// TwinCAT 3 PLC project SAT_Bibliothek
// Title: STOBER_G6_Util
// Company: STÖBER Antriebstechnik GmbH + Co. KG
// Author: STOBER
// ProjectVersion: 3.1.1.0
// Description: The function blocks in the library would be operational with STOBER drive controller Firmware version 6.5-F and higher.
// ProgramVersion: 3.1.4024.12
// libraries:
//   Tc2_EtherCAT, * (Beckhoff Automation GmbH)
//   Tc2_MC2, * (Beckhoff Automation GmbH)
//   Tc2_MC2_Drive, * (Beckhoff Automation GmbH)
//   Tc2_Standard, * (Beckhoff Automation GmbH)
//   Tc2_System, * (Beckhoff Automation GmbH)
//   Tc2_Utilities, * (Beckhoff Automation GmbH)
//   Tc3_Module, * (Beckhoff Automation GmbH)
// project tree:
//   DUTs/STOBER_Backup_Restore/ eFBERROR.TcTLEO, eSERVICE.TcTLEO, eWriteState.TcTLEO, E_EventType.TcTLEO, ST_DeviceInfo.TcDUT, ST_Event.TcDUT
//   DUTs/STOBER_Boxname/ Ethercat_State.TcDUT, StoeberSlavedesc.TcDUT, St_Error.TcDUT
//   DUTs/STOBER_MC_HOME/ eERROR.TcTLEO, st_Set_Value.TcDUT
//   GVLs/ GLOBAL_DeviceInfo.TcGVL, GVL_Constant.TcGVL
//   POUs/ FB_STOBER_BASE.TcPOU, STOBER_Backup_Restore.TcPOU, STOBER_BoxName.TcPOU, STOBER_MC_HOME.TcPOU
//   POUs/Functions/ CONCAT4.TcPOU, CONCAT8.TcPOU
//   POUs/Logger/ FB_logger.TcPOU, FB_LogPersistentStorage.TcPOU, GetSystemTimeStamp.TcPOU, I_PersistentEventStorage.TcIO
//   Project Information/ F_GetCompany.TcPOU, F_GetTitle.TcPOU, F_GetVersion.TcPOU
//   Version/ Global_Version.TcGVL

// ---- DUTs/STOBER_Backup_Restore/eFBERROR.TcTLEO
{attribute 'qualified_only'}
{attribute 'strict'}
TYPE eFBERROR :
(   
	(*Function block errors*)
	NoError								:=0,
	WrongFilePath						:=101,
	WrongDS6_ProcessPath				:=103,
	WrongEtherCATRevision				:=105,
	InvalidBoxname						:=107,
	WrongServiceTypeInput				:=109,
	TimeoutExceed						:=111,
	NoStoberSlaveInConfiguration		:=113,
	
	(*DS6 Errors*)
	ProjectNotFound						:=201,//Drive controller project not found
	MoreThanOneProjectFound				:=203,//Drive Controller found several times in project 
	OpenProjectError					:=205,//project open error 
	ConnectionError						:=207,//Connection to Drive controller failed 
	OnlineError							:=209//Online connection failed 
	
	


);
END_TYPE

// ---- DUTs/STOBER_Backup_Restore/eSERVICE.TcTLEO
{attribute 'qualified_only'}
{attribute 'strict'}
TYPE eSERVICE :
(
	Backup			:=0,
	Backup_RevDocu	:=1,
	Restore			:=2

);
END_TYPE

// ---- DUTs/STOBER_Backup_Restore/eWriteState.TcTLEO
{attribute 'qualified_only'}
{attribute 'strict'}
{attribute  'hide'}
TYPE eWriteState :
(
	FileOpen_TRIGGER,
	FILE_OPEN,
	WAIT_FOR_EVENT,
	WRITE_EVENT_TRIGGER,
	WRITE_EVENT,
	FILE_CLOSE_TRIGGER,
	FILE_CLOSE,ERROR
);
END_TYPE

// ---- DUTs/STOBER_Backup_Restore/E_EventType.TcTLEO
{attribute 'qualified_only'}
{attribute 'strict'}
{attribute 'to_string'}
{attribute  'hide'}
TYPE E_EventType :
(
	Info:=0,
	Warning:=1,
	Error:=2
);
END_TYPE

// ---- DUTs/STOBER_Backup_Restore/ST_DeviceInfo.TcDUT
{attribute  'hide'}
TYPE ST_DeviceInfo :
STRUCT
	Slave_Address		:STRING(16);
	Production_Number	:STRING(16);
END_STRUCT
END_TYPE

// ---- DUTs/STOBER_Backup_Restore/ST_Event.TcDUT
{attribute  'hide'}
TYPE ST_Event :
STRUCT
	EventType:T_MaxString;
	sEventText:T_MaxString;
	timesatamp:T_MaxString;
END_STRUCT
END_TYPE

// ---- DUTs/STOBER_Boxname/Ethercat_State.TcDUT
{attribute 'qualified_only'}
{attribute 'strict'}
{attribute 'hide'}
TYPE Ethercat_State :
(
	INIT :=1,
	PREOP:=2,
	SAFEOP:=4,
	OP:=8
);
END_TYPE

// ---- DUTs/STOBER_Boxname/StoeberSlavedesc.TcDUT
{attribute 'hide'}
TYPE StoeberSlavedesc :
STRUCT
	nAddr:WORD;
	sType:STRING(15);
	{attribute 'TcEncoding' := 'UTF-8'}
	sName:STRING(31);
	nDevType:DWORD;
	iState:INT;
END_STRUCT
END_TYPE

// ---- DUTs/STOBER_Boxname/St_Error.TcDUT
{attribute 'hide'}
TYPE St_Error :
STRUCT
	
END_STRUCT
END_TYPE

// ---- DUTs/STOBER_MC_HOME/eERROR.TcTLEO
{attribute 'qualified_only'}
{attribute 'strict'}
TYPE eERROR :
(
	NO_ERROR := 0, //Defined operation was executed successfully
	HOMING_METHOD_INACTIVE:=1,//NO homing method selected 
	AXIS_NOT_ENABLED:=2,//Axis is not enabled 
	WRONG_MODE:=3,//Wrong mode of operation input 
	NO_DEVICE_LINK:=4//ModeOfOperation output variable is not linked in device config  
);
END_TYPE

// ---- DUTs/STOBER_MC_HOME/st_Set_Value.TcDUT
{attribute 'hide'}
TYPE st_Set_Value :
STRUCT
	SetPosition		:LREAL;
	SetVelocity		:LREAL;
	SetAcc			:LREAL;
	SetDec			:LREAL;
	SetDirection	:LREAL;
	SetJerk			:LREAL;
END_STRUCT
END_TYPE

// ---- GVLs/GLOBAL_DeviceInfo.TcGVL
{attribute 'qualified_only'}
VAR_GLOBAL
	arr_DeviceInfodata:ARRAY [1..GVL_Constant.MAX_STOBER_SLAVES] OF ST_DeviceInfo;
END_VAR

// ---- GVLs/GVL_Constant.TcGVL
{attribute 'qualified_only'}
VAR_GLOBAL CONSTANT
	MAX_STOBER_SLAVES:INT:=200;
	MaxSlaves:INT:=2000;
END_VAR

// ---- Version/Global_Version.TcGVL
{attribute 'TcGenerated'}
{attribute 'no-analysis'}
{attribute 'linkalways'}
// This function has been automatically generated from the project information.
VAR_GLOBAL CONSTANT
	{attribute 'const_non_replaced'}
	stLibVersion_STOBER_G6_Util : ST_LibVersion := (iMajor := 3, iMinor := 1, iBuild := 1, iRevision := 0, nFlags := 0, sVersion := '3.1.1.0');
END_VAR

// ---- POUs/Logger/I_PersistentEventStorage.TcIO
INTERFACE I_PersistentEventStorage

METHOD StoreEvent 
VAR_INPUT
	stEvent:ST_Event;
END_VAR
END_METHOD

END_INTERFACE

// ---- POUs/FB_STOBER_BASE.TcPOU
FUNCTION_BLOCK ABSTRACT FB_STOBER_BASE
VAR
	
END_VAR

METHOD GetInstanceName : T_MAXSTRING
VAR_INPUT
END_VAR
VAR_INPUT
	Str1:T_MaxString;
END_VAR
VAR
	ptByte		:POINTER TO BYTE;
	ptDestByte	:POINTER TO BYTE;
	Ret_String	:T_MaxString;
	ptrRtnByte	:POINTER TO BYTE;
	i			:INT;
	count		:INT;
	arrBytes		:ARRAY [0..255] OF BYTE;
	j			:UINT;
END_VAR
VAR CONSTANT
	CHAR_DOT:INT:=46;//the ascii code for '.' character
END_VAR
//set the initial adress 
ptByte:=ADR(Str1);
ptDestByte:=ptByte;
//reset the Array of byte 
FOR j:=0 TO 255 DO 
	arrBytes[j]:=0;
END_FOR
ptrRtnByte:=ADR(arrBytes);//set initial adress 

count:=0;
FOR i:=0 TO LEN(Str1) DO 
	IF ptDestByte^<>0 THEN
		//save the string
		IF ptDestByte^=CHAR_DOT THEN //check for '.' character 
			count:=count+1;
		END_IF 
		IF count>=2 THEN
			IF count=2 AND  ptDestByte^=CHAR_DOT THEN 
				ptDestByte:=ptDestByte+1;
			END_IF
			ptrRtnByte^:=ptDestByte^;//here start with Main.Fb1.variableName
			ptrRtnByte:=ptrRtnByte+1;
		END_IF
		ptDestByte:=ptDestByte+1;
	END_IF
END_FOR

GetInstanceName:=BYTEARR_TO_MAXSTRING(arrBytes);
END_METHOD

END_FUNCTION_BLOCK

// ---- POUs/Functions/CONCAT4.TcPOU
FUNCTION CONCAT4 : T_MaxString
VAR_INPUT
	STR1	:T_MaxString;
	STR2	:T_MaxString;
	STR3	:T_MaxString;
	STR4	:T_MaxString;
END_VAR
VAR
	_MainString	:T_MaxString:='';
END_VAR

_MainString:=CONCAT(STR1:=STR1,STR2:=STR2);
_MainString:=CONCAT(STR1:=_MainString,STR2:=STR3);
_MainString:=CONCAT(STR1:=_MainString,STR2:=STR4);

CONCAT4:=_MainString;

END_FUNCTION

// ---- POUs/Functions/CONCAT8.TcPOU
FUNCTION CONCAT8 : T_MaxString
VAR_INPUT
	STR1	:T_MaxString;
	STR2	:T_MaxString;
	STR3	:T_MaxString;
	STR4	:T_MaxString;
	STR5	:T_MaxString;
	STR6	:T_MaxString;
	STR7	:T_MaxString;
	STR8	:T_MaxString;
END_VAR
VAR
	_MainString	:T_MaxString:='';
END_VAR

_MainString:=CONCAT(STR1:=STR1,STR2:=STR2);
_MainString:=CONCAT(STR1:=_MainString,STR2:=STR3);
_MainString:=CONCAT(STR1:=_MainString,STR2:=STR4);
_MainString:=CONCAT(STR1:=_MainString,STR2:=STR5);
_MainString:=CONCAT(STR1:=_MainString,STR2:=STR6);
_MainString:=CONCAT(STR1:=_MainString,STR2:=STR7);
_MainString:=CONCAT(STR1:=_MainString,STR2:=STR8);

CONCAT8:=_MainString;

END_FUNCTION

// ---- POUs/Logger/FB_logger.TcPOU
FUNCTION_BLOCK FB_logger
VAR
	_fbGetLocalTime		:FB_LocalSystemTime;
	_TimeStampNow		:STRING;
	_logmessage			:T_MaxString;
	_StEvent			:ST_Event;
	_PersistentStorage  :I_PersistentEventStorage;
END_VAR

METHOD PUBLIC AddEvent : BOOL
VAR_INPUT
	 EventType:T_MaxString;
	//EventSeverity:TcEventSeverity;
	//nEventIdentity:UINT;
	sEventText:T_MaxString;
END_VAR
VAR
	_TrigEvent:R_Trig;
END_VAR
//Assign event structure 
_StEvent.EventType:=EventType;
_StEvent.sEventText:=sEventText;
GetSystemTimeStamp(stEvent:=_StEvent);

//Call storage event 
_PersistentStorage.StoreEvent(stEvent:=_StEvent);
END_METHOD

METHOD FB_init : BOOL
VAR_INPUT
	bInitRetains : BOOL; // if TRUE, the retain variables are initialized (warm start / cold start)
	bInCopyCode : BOOL;  // if TRUE, the instance afterwards gets moved into the copy code (online change)
	iPersitentstorage:I_PersistentEventStorage;
END_VAR
_PersistentStorage:=iPersitentstorage;
END_METHOD

END_FUNCTION_BLOCK

// ---- POUs/Logger/GetSystemTimeStamp.TcPOU
FUNCTION GetSystemTimeStamp
VAR_INPUT
	stEvent:REFERENCE TO ST_Event;
END_VAR
VAR
	fbGetSYSTEMTIME			:	GETSYSTEMTIME;
	stFileTime				:	T_FILETIME;
	dateNow					:   T_MAXSTRING;
	timeNow					:	T_MaxString;
	fbFiletime_toLocaltime	:	FB_FileTimeToTzSpecificLocalTime;
END_VAR

fbGetSYSTEMTIME(timeLoDW=>stFileTime.dwLowDateTime,
				timeHiDW=>stFileTime.dwHighDateTime);
				
//Specific local time in WEST europe zone--Daylight saving time 
fbFiletime_toLocaltime(in:=stFileTime,tzInfo:=WEST_EUROPE_TZI);		
				
dateNow:=REPLACE(TO_STRING(TO_DATE(FILETIME_TO_DT(fbFiletime_toLocaltime.out))),'',2,1);	//Replace D#YYYY-MM-DD with YYYY-MM-DD			
TimeNow:=REPLACE(TO_STRING(DT_TO_TOD(FILETIME_TO_DT(fbFiletime_toLocaltime.out))),'',4,1); //Replace TOD#HH:MM:SS with HH:MM:SS
stEvent.timesatamp:=CONCAT(CONCAT(dateNow,'  '),timeNow);

END_FUNCTION

// ---- POUs/Logger/FB_LogPersistentStorage.TcPOU
FUNCTION_BLOCK FB_LogPersistentStorage IMPLEMENTS I_PersistentEventStorage
VAR_INPUT
	sPathName			:STRING;
END_VAR
VAR_OUTPUT
	Error				:BOOL;
END_VAR
VAR
	fbFileOpen			:FB_FileOpen;
	fbFilePuts			:FB_FilePuts;
	fbFileClose			:FB_FileClose;
	eLogWriteState		:eWriteState;
	stEventWriteToFile	:ST_Event;
	csvString			:T_MaxString;
END_VAR

CASE eLogWriteState OF 
	eWriteState.FileOpen_TRIGGER://open file
		fbFileOpen(sNetId:='',nMode:=FOPEN_MODEAPPEND OR FOPEN_MODETEXT,
					sPathName:=sPathName,ePath:=PATH_GENERIC,bExecute:=TRUE);
		IF NOT fbFileOpen.bBusy THEN 
			IF fbFileOpen.bError THEN
				eLogWriteState:=eWriteState.ERROR;
			ELSE
				fbFileOpen(sNetId:='',bExecute:=FALSE);
				eLogWriteState:=eWriteState.WAIT_FOR_EVENT;
			END_IF
		END_IF 			
				
  
	eWriteState.WAIT_FOR_EVENT:
		//do nothing here waits for the event to trigger the new event see the store event 
		
	eWriteState.WRITE_EVENT_TRIGGER:
		csvString:=CreateLogString(stEvent:=stEventWriteToFile);
		fbFilePuts(sNetId:='',bExecute:=TRUE,sLine:=csvString,hFile:=fbFileOpen.hFile);
		IF NOT fbFilePuts.bBusy THEN 
			IF fbFilePuts.bError THEN
				eLogWriteState:=eWriteState.ERROR;
			ELSE
				fbFilePuts(sNetId:='',bExecute:=FALSE);
				eLogWriteState:=eWriteState.FILE_CLOSE_TRIGGER;
			END_IF
		END_IF
		
	eWriteState.FILE_CLOSE_TRIGGER:
		fbFileClose(bExecute:=TRUE,hFile:=fbFileOpen.hFile);
		IF NOT fbFileClose.bBusy THEN 
			IF fbFileClose.bError THEN
				eLogWriteState:=eWriteState.ERROR;
			ELSE
				fbFileClose(sNetId:='',bExecute:=FALSE);
				eLogWriteState:=eWriteState.FileOpen_TRIGGER;
			END_IF
		END_IF
		
	eWriteState.ERROR:
		Error:=TRUE;

END_CASE

METHOD PRIVATE CreateLogString : T_MaxString
VAR_INPUT
	stEvent:REFERENCE TO ST_Event;
END_VAR
VAR 
	tempString:T_MaxString;
END_VAR
tempString:=stEvent.timesatamp;
tempString:=CONCAT(CONCAT(tempString,' : '),(stEvent.EventType));
tempString:=CONCAT(CONCAT(tempString,' : '),stEvent.sEventText);
tempString:=CONCAT(tempString,'$N');
CreateLogString:=tempString;
END_METHOD

METHOD StoreEvent
VAR_INPUT
	stEvent	: ST_Event;
END_VAR
IF eLogWriteState=eWriteState.WAIT_FOR_EVENT THEN 
	eLogWriteState:=eWriteState.WRITE_EVENT_TRIGGER;
	stEventWriteToFile:=stEvent;
END_IF
END_METHOD

END_FUNCTION_BLOCK

// ---- POUs/STOBER_Backup_Restore.TcPOU
{attribute 'reflection'}
FUNCTION_BLOCK STOBER_Backup_Restore EXTENDS FB_STOBER_BASE
VAR_INPUT
	Execute						:BOOL;				//Activation of function block by a rise edge at this input 
	AmsNetId_EtherCAT_Master	:T_AmsNetID;		//AMS network ID of the EtherCAT master device 
	Filepath					:T_MAXSTRING;		//
	DS6_ProcessPath				:T_MAXSTRING; 		//
	Slave_addr					:UINT;				//Adress of the EtherCAT slave(Stober Drive controller)
	Servicetype					:eSERVICE;			//Requested service Backup/restore 
END_VAR
VAR_OUTPUT
	Done						:BOOL;
	Busy						:BOOL;
	Error						:BOOL;
	nErrId_ADS					:UDINT;
	nFbErrorID					:eFBERROR;
	InitDone					:BOOL;	
	iAction						:INT;
END_VAR
VAR	
	init								:BOOL;
	_nState_FileHandle					:INT;
	_iState								:INT;
	
	_fbGetSlaveIdentity					:FB_EcGetSlaveIdentity;//Function block return EtherCAT slave identity (vendor-id,serialNr,EtherCAT revision etc)
	_fbFileOpen							:FB_FileOpen;//Function block to open the file
	_fbFileClose						:FB_FileClose;//Function block to close the file
	_fbFileGets							:FB_FileGets;//Reads the file line by line
	_fbFileWrite						:FB_FileWrite; //Function block to write the file 
	_newFileCreated						:BOOL;
	_fbCOESdoRead,fbSdoReadBoxName		:FB_EcCoESdoRead;//function block to read DS6 parameter over EtherCAT sdo
	_readDriveControllerProductionNr						:STRING(16);//Produnction number of the Drive controller
	_hFile								:UINT; //File header
	_bEOF								:BOOL;//End of file status 
	_Synchronous_flag  					:DWORD; //ADS return value 
	_FbLogPersitentStorage				:FB_LogPersistentStorage;//store the log data 
	_fbLogger							:FB_logger(_FbLogPersitentStorage);
	_EventTrigger						:R_TRIG;
	_ActivateNTProcess					:NT_StartProcess;
	{attribute 'instance-path'} 
    {attribute 'noinit'} 
	_spath								:T_MaxString;
	_subindex							:BYTE;
	_oldProductionNr					:STRING;
	 //{attribute 'TcEncoding':='UTF-8'}
	_sBoxName							:STRING(79);
	_sBoxNameUTF_8						:STRING;
	_ErrorMessage						:STRING;
	_fbTimeOut							:TON;
	
	_fbExecuteTrig						:R_TRIG;
	_CommandLine						:T_MaxString;
	_eventText							:T_MaxString;
	_BackupRestoreTrig					:R_Trig;
	_projectPath						:STRING;
	_initError							:BOOL;
	_initFbErrorID						:eFBERROR;
	_initADSErrorID						:UDINT;
	_ErrorState							:INT;
	_initErrorState						:INT;
	_deviceDescPath						:T_MaxString;
	_fbFilepath_EnumFindFileEntry		:FB_EnumFindFileEntry;
	_fbDS6ProcessPath_EnumFindFileEntry	:FB_EnumFindFileEntry;
	_filepathexists						:BOOL;
	_indexArray							:INT:=1;
	_StoreArrayIndex					:INT;
	_FileWriteByteArray					:ARRAY [0..MAX_BYTEARRAY_SIZE] OF BYTE;
	_newSlave_In_Topology				:BOOL;
	_xFirstInvocation					:BOOL;
	_fbCreateDir						:FB_CreateDir;
END_VAR

VAR CONSTANT
	MAX_BYTEARRAY_SIZE:INT:=4000;
END_VAR

//_prouctionNr als _readDriveControllerProductionNr

(********************************************Method calls and initialisation of the function blocks************************************)
(*Author--Anuj Sambhare*)
(*log-method call*)
(*initialise devicedescription file path *)
_fbExecuteTrig(CLK:=Execute);

IF _filepathexists THEN 
	_FbLogPersitentStorage(sPathName:=CONCAT(Filepath,'\log\Tc_Log.log'));
	_fbLogger();
	_deviceDescPath:=CONCAT(Filepath,'\DeviceInfo.txt');
END_IF

(*call Outputhandle--- Function block output variables handling *)

OutputHandle();

(*method call to call the internal function blocks used.*)
CallInternalFbs();

(*Method call for Backup and restore execution *)
(*
IF NOT _initError AND  init AND _fbExecuteTrig.Q THEN 
	init:=FALSE;
END_IF
*)

BackupRestore();

//Reinit after exectute 
(*
IF  _fbExecuteTrig.Q AND init THEN 
	init:=FALSE;
	_nState_FileHandle:=0;
END_IF
*)
IF init THEN 
	InitDone:=TRUE;
ELSE
	InitDone:=FALSE;	
END_IF

	
IF NOT init THEN
	(*Read the Production Number*) 	
	CASE _nState_FileHandle OF 
		0:
			(*check if project path exits  (Als Method erstellen*)
			_fbFilepath_EnumFindFileEntry(bExecute:=TRUE);
			IF NOT _fbFilepath_EnumFindFileEntry.bBusy THEN 
				IF _fbFilepath_EnumFindFileEntry.bError THEN 
					Error:=TRUE;
					_fbFilepath_EnumFindFileEntry(bExecute:=FALSE);
					_initErrorState:=_nState_FileHandle;
					_nState_FileHandle:=999;
					_initADSErrorID:=_fbFilepath_EnumFindFileEntry.nErrID;
				ELSIF _fbFilepath_EnumFindFileEntry.stFindFile.sFileName<> '' THEN 
					_filepathexists:=TRUE;
					_fbCreateDir(sNetId:='',sPathName:=CONCAT(Filepath,'\log'),ePath:=E_OpenPath.PATH_GENERIC,bExecute:=TRUE);
					_nState_FileHandle:=1;	
					_fbFilepath_EnumFindFileEntry(bExecute:=FALSE); 
				ELSE 
					_fbFilepath_EnumFindFileEntry(bExecute:=FALSE);
					Error:=TRUE;
					_initErrorState:=_nState_FileHandle;
					(*fehler code 101*)
					_initFbErrorID:=eFBERROR.WrongFilePath;
					_nState_FileHandle:=999;	
				END_IF
			END_IF
		
		1:
			(*check if ds6 process path (Als Method erstellen*)
			_fbDS6ProcessPath_EnumFindFileEntry(bExecute:=TRUE);
			IF NOT _fbDS6ProcessPath_EnumFindFileEntry.bBusy THEN 
				IF _fbDS6ProcessPath_EnumFindFileEntry.bError THEN 
					Error:=TRUE;
					_fbDS6ProcessPath_EnumFindFileEntry(bExecute:=FALSE);
					_initADSErrorID:=_fbDS6ProcessPath_EnumFindFileEntry.nErrID;
					_initErrorState:=_nState_FileHandle;
					_nState_FileHandle:=999;
				ELSIF _fbDS6ProcessPath_EnumFindFileEntry.stFindFile.sFileName<> '' THEN 
					_nState_FileHandle:=2;	
					_fbDS6ProcessPath_EnumFindFileEntry(bExecute:=FALSE); 
				ELSE 
					_fbDS6ProcessPath_EnumFindFileEntry(bExecute:=FALSE);
					Error:=TRUE;
					_initErrorState:=_nState_FileHandle;
					(*Fehler code 103*)
					_initFbErrorID:=eFBERROR.WrongDS6_ProcessPath;
					_nState_FileHandle:=999;	
				END_IF
			END_IF
	
		2:(*Read EtherCAT slave identity revision*) 
		  (*later on change with FB_EcGetSlaveIdentity, no dependancy on EtherCAT states*)
		  (*This case is only programmed in order to get the ethercat revision number because at the moment the production number
		    of the drive controller is not saved in the EEPROM.*) 
			_EventTrigger(CLK:=FALSE);
			_fbGetSlaveIdentity(sNetId:=AmsNetId_EtherCAT_Master,nSlaveAddr:=Slave_addr,
								bExecute:=TRUE);
			IF NOT _fbGetSlaveIdentity.bBusy THEN 
				IF _fbGetSlaveIdentity.bError THEN 
					_fbGetSlaveIdentity(bExecute:=FALSE);	
						_initADSErrorID:=_fbGetSlaveIdentity.nErrId;
						Error:=TRUE;
						_initErrorState:=_nState_FileHandle;
						_ErrorMessage:=CONCAT4(STR1:=GetInstanceName(_spath),STR2:=' ',STR3:='GetSlaveIdentity ADS Error ',STR4:=TO_STRING(_initADSErrorID));
						_nState_FileHandle:=999;
				ELSE
					_fbGetSlaveIdentity(bExecute:=FALSE);
					IF _fbGetSlaveIdentity.identity.revisionNo=6500 THEN 
						_subindex:=16#3;
						_nState_FileHandle:=3;
					ELSIF _fbGetSlaveIdentity.identity.revisionNo=6000 THEN 
						_subindex:=16#3;
						_nState_FileHandle:=3;
					ELSIF _fbGetSlaveIdentity.identity.revisionNo=6100 THEN 
						_subindex:=16#2;
						_nState_FileHandle:=3;	
					ELSE
						Error:=TRUE;
						_ErrorMessage:='Wrong etherCAT template revision.';
						_initErrorState:=_nState_FileHandle;
						(*Fehler code 105*)
						_initFbErrorID:=eFBERROR.WrongEtherCATRevision;
						_nState_FileHandle:=999;	
					END_IF
				END_IF
			END_IF					
	
		3:
			(*read the production number index number for parameter E52[2](Production number)=16#2834*) 			
			_fbCOESdoRead(sNetId:=AmsNetId_EtherCAT_Master,nSlaveAddr:=Slave_addr ,nSubIndex:=_subindex,nIndex:=16#2834 , 
						pDstBuf:=ADR(_readDriveControllerProductionNr),cbBufLen:=SIZEOF(_readDriveControllerProductionNr) ,bExecute:=TRUE );
			IF NOT _fbCOESdoRead.bBusy THEN 
				IF _fbCOESdoRead.bError THEN 
					_ErrorMessage:='';
					_fbCOESdoRead(bExecute:=FALSE);
					_initADSErrorID:=_fbCOESdoRead.nErrId;
					_ErrorMessage:=CONCAT4(STR1:=GetInstanceName(_spath),STR2:=' ',STR3:='EtherCAT Sdo Read  ADS Error ',STR4:=TO_STRING(_initADSErrorID));
					Error:=TRUE;(*Generate log*) 
					_initErrorState:=_nState_FileHandle;
					_nState_FileHandle:=999;
				ELSE
					_fbCOESdoRead(bExecute:=FALSE);	
					_nState_FileHandle:=4;
				END_IF
			END_IF
			
		4:
			_indexArray:=1;
			_nState_FileHandle:=5;
			
			
		5:	(*check if file exists*) 
			(*if file doesnt exist in the directory then Function block will show 1804 error*) 
			_fbFileOpen(sNetId:='' ,sPathName:=_deviceDescPath ,nMode:=FOPEN_MODEREAD ,ePath:=PATH_GENERIC ,bExecute:=TRUE , hFile=>_hFile );
			IF NOT _fbFileOpen.bBusy THEN 
				IF (_hFile=0 AND _fbFileOpen.nErrId=1804) THEN (*Error 1804 comes when file is in read mode and the file does not exist project folder*)				 
					_fbFileOpen(sNetId:='',bExecute:=FALSE);
					_nState_FileHandle:=6;(*Go to state 6 to create a new file*)
			    ELSIF (_fbFileOpen.nErrId<>1804 AND _fbFileOpen.bError) THEN
					_fbFileOpen(sNetId:='',bExecute:=FALSE);
					_ErrorMessage:='';
					Error:=TRUE;
					_initErrorState:=_nState_FileHandle;
					_initADSErrorID:=_fbFileOpen.nErrId;
					_ErrorMessage:=CONCAT4(STR1:=GetInstanceName(_spath),STR2:=' ',STR3:='File open ADS Error ',STR4:=TO_STRING(_initADSErrorID));
					_nState_FileHandle:=999;(*Generate log*) 
				ELSE (*File already exist go to step 50 to read the production number *)
					_fbFileOpen(sNetId:='',bExecute:=FALSE);
					_nState_FileHandle:=50;
				END_IF	
			END_IF
			
		6:(*create new deviceinfo.txt file*) 
			_fbFileOpen(sNetId:='',sPathName:=_deviceDescPath ,nMode:=FOPEN_MODEAPPEND OR FOPEN_MODETEXT ,ePath:=PATH_GENERIC ,bExecute:=TRUE , hFile=>_hFile );
			IF NOT _fbFileOpen.bBusy THEN 
				IF _fbFileOpen.bError THEN 
					_ErrorMessage:='';
					_fbFileOpen(sNetId:='',bExecute:=FALSE);
					Error:=TRUE;(*Generate log*) 
					_initErrorState:=_nState_FileHandle;
					_initADSErrorID:=_fbFileOpen.nErrId;
					_ErrorMessage:=CONCAT4(STR1:=GetInstanceName(_spath),STR2:=' ',STR3:='File Open ADS Error ',STR4:=TO_STRING(_initADSErrorID));
					_nState_FileHandle:=999;
				ELSE
					_fbFileOpen(sNetId:='',bExecute:=FALSE);
					_nState_FileHandle:=7;	
				END_IF
			END_IF
			
		7:(*close the file without inserting the data*) 
			_fbFileClose(sNetId:='',hFile:=_hFile,bExecute:=TRUE);
			IF NOT _fbFileClose.bBusy THEN 
				IF _fbFileClose.bError THEN 
					Error:=TRUE;
					_initErrorState:=_nState_FileHandle;
					_initADSErrorID:=_fbFileClose.nErrId;
					_ErrorMessage:=CONCAT4(STR1:=GetInstanceName(_spath),
									STR2:=' ',STR3:='File close ADS Error ',STR4:=TO_STRING(_initADSErrorID));
					_fbFileClose(sNetId:='',bExecute:=FALSE);					
					_nState_FileHandle:=999;
				ELSE
					_fbFileClose(sNetId:='',bExecute:=FALSE);	
					_nState_FileHandle:=30;
					iAction:=2;
				END_IF
			END_IF
		
		30:(*New file DeviceInfo.txt is created in the filepath directory*)
			_newFileCreated:=TRUE;
			init:=TRUE;
			
		50:(*Open deviceinfo.txt file*)
			_newFileCreated:=FALSE;
			 _fbFileOpen(sNetId:='' ,sPathName:=_deviceDescPath ,nMode:=FOPEN_MODEREAD OR FOPEN_MODETEXT,
						ePath:=PATH_GENERIC,bExecute:=TRUE,hFile=>_hFile);
					
			IF NOT _fbFileOpen.bBusy THEN 
				IF _fbFileOpen.bError THEN 
					_fbFileOpen(sNetId:='',bExecute:=FALSE);
					_initADSErrorID:=_fbFileOpen.nErrId;
					_ErrorMessage:=CONCAT4(STR1:=GetInstanceName(_spath),STR2:=' ',
											STR3:='ADS Error ',STR4:=TO_STRING(_initADSErrorID));
					Error:=TRUE;
					_initErrorState:=_nState_FileHandle;
					_nState_FileHandle:=999;
				ELSE
					_fbFileOpen(sNetId:='',bExecute:=FALSE);
					_nState_FileHandle:=60;
				END_IF
			END_IF
			
		 60:(*Read the file line by line*)	
			_fbFileGets(sNetId:='',bExecute:=TRUE,hFile:=_hFile,bEOF=>_bEOF);
			IF NOT _fbFileGets.bBusy THEN 
				IF _fbFileGets.bError THEN 
					Error:=TRUE;
					_initErrorState:=_nState_FileHandle;
					_initADSErrorID:=_fbFileGets.nErrId;
					_ErrorMessage:=CONCAT4(STR1:=GetInstanceName(_spath),STR2:=' ',
										   STR3:='File readline ADS Error ',STR4:=TO_STRING(_initADSErrorID));
					_fbFileGets(bExecute:=FALSE);
					_nState_FileHandle:=999;
				ELSE
					_fbFileGets(sNetId:='',bExecute:=FALSE);
					_nState_FileHandle:=70;
				END_IF
			END_IF
		
			
		70:
			IF _indexArray<GVL_Constant.MAX_STOBER_SLAVES THEN 
				IF NOT _bEOF THEN  		
					GLOBAL_DeviceInfo.arr_DeviceInfodata[_indexArray].Slave_Address:=GetSlaveAddress(Str1:=_fbFileGets.sLine);
					GLOBAL_DeviceInfo.arr_DeviceInfodata[_indexArray].Production_Number:=GetProductionNumber(Str1:=_fbFileGets.sLine);
					_indexArray:=_indexArray+1;
					_nState_FileHandle:=60;
			    ELSE
						_nState_FileHandle:=80;	
				END_IF	
			END_IF
		
			
			
		80:	(*Prepare array data*)
			FOR _indexArray:=1 TO GVL_Constant.MAX_STOBER_SLAVES DO 
				IF GLOBAL_DeviceInfo.arr_DeviceInfodata[_indexArray].Slave_Address=TO_STRING(Slave_addr) THEN
					    (*compare the production number*)
						_newSlave_In_Topology:=FALSE;
						IF TO_STRING(GLOBAL_DeviceInfo.arr_DeviceInfodata[_indexArray].Production_Number)=_readDriveControllerProductionNr THEN 
							iAction:=0;
							_nState_FileHandle:=90;
						ELSE
							iAction:=2;
							_nState_FileHandle:=100;
						END_IF
					EXIT;	
				END_IF
				IF _indexArray>=GVL_Constant.MAX_STOBER_SLAVES THEN 
					iAction:=2;
					_newSlave_In_Topology:=TRUE;
					_nState_FileHandle:=140;	
				END_IF
			END_FOR
			
		90:(*Production number exists ready for backup close the file*)
			_fbFileClose(sNetId:='',hFile:=_hFile,bExecute:=TRUE);
			IF NOT _fbFileClose.bBusy THEN 
				IF _fbFileClose.bError THEN 
					_initADSErrorID:=_fbFileClose.nErrId;
					_ErrorMessage:=CONCAT4(STR1:=GetInstanceName(_spath),STR2:=' ',
											STR3:='File close ADS Error ',STR4:=TO_STRING(_initADSErrorID));
					Error:=TRUE;
					_initErrorState:=_nState_FileHandle;
					_fbFileClose(sNetId:='',bExecute:=FALSE);	
					_nState_FileHandle:=999;
				ELSE
					_fbFileClose(sNetId:='',bExecute:=FALSE);	
					_nState_FileHandle:=140;
				END_IF
			END_IF
		
		100:(*Close the deviceinfo.txt file first if production nr does not exist*)
			iAction:=2;	(*Restore is needed *)
			_fbFileClose(sNetId:='',hFile:=_hFile,bExecute:=TRUE);
			IF NOT _fbFileClose.bBusy THEN 
				IF _fbFileClose.bError THEN 
					_initADSErrorID:=_fbFileClose.nErrId;
					_ErrorMessage:=CONCAT4(STR1:=GetInstanceName(_spath),STR2:=' ',
											STR3:='File close ADS Error ',STR4:=TO_STRING(_initADSErrorID));
					Error:=TRUE;
					_initErrorState:=_nState_FileHandle;
					_fbFileClose(sNetId:='',bExecute:=FALSE);	
					_nState_FileHandle:=999;
				ELSE
					_fbFileClose(sNetId:='',bExecute:=FALSE);	
					_nState_FileHandle:=140;
				END_IF
			END_IF
			
			
		140:(*Production number and slave address does not exit*)
			init:=TRUE;	
			
		300:(*Production number already exists*)			
			init:=TRUE;
			
		999:(*Error case*)
			 _initError:=TRUE;
			 Error:=_initError;
			 _EventTrigger(CLK:=TRUE);
			IF _EventTrigger.Q THEN 
				_fbLogger.AddEvent(sEventText:=_ErrorMessage,EventType:='Error');
			END_IF		
			init:=TRUE;		
	END_CASE
END_IF

(*Method Activate the subprocess*)
METHOD PRIVATE ActivateProcess : BOOL

VAR
	_fbWaitTimer:TON;
END_VAR
(*Method activates the NT_StartProcess function block to start a Drive Control Suite application with a commandline for project read or write*)
(*Start DS6 applicationfrom TwinCAT
Commandline=> DS6.exe --command <command> --boxname <Boxname> --productionnumber <number> --projectpath <path> --instancename <name>
*) 
 _ActivateNTProcess(START:=TRUE);

IF NOT _ActivateNTProcess.BUSY THEN 
	IF _ActivateNTProcess.ERR THEN 
		Error:=TRUE;
		_ErrorState:=_iState;
		nErrId_ADS:=_ActivateNTProcess.ERRID;
		_eventText:=Concat4(STR1:=GetInstanceName(_spath),STR2:=' ',STR3:='NTProcess ADS Error ',STR4:=TO_STRING(nErrId_ADS));
		_EventTrigger(CLK:=TRUE);		
		IF _EventTrigger.Q THEN 
			_fbLogger.AddEvent(sEventText:=_eventText,EventType:='Error');
			_EventTrigger(CLK:=FALSE);	
		END_IF	
		_ActivateNTProcess(START:=FALSE);
		_iState:=99;						
	ELSE
		_ActivateNTProcess(START:=FALSE);
		_iState:=_iState+1;							
	END_IF							
END_IF
END_METHOD

METHOD PRIVATE BackupRestore : BOOL
VAR
	i: INT;
END_VAR

_fbTimeOut(PT:=SetTimeout());


CASE _iState OF
 
	0://Execute 	
		IF _fbExecuteTrig.Q  THEN 
			busy:=TRUE;
			Done:=FALSE;
			_Synchronous_flag:=0;
			Error:=FALSE;
			
			nErrId_ADS:=0;
			nFbErrorID:=0;
			_ErrorMessage:='';
			_fbTimeOut.IN:=FALSE;
			_EventTrigger(CLK:=FALSE);
			_BackupRestoreTrig(CLK:=FALSE);
			_nState_FileHandle:=0;
			init:=FALSE;			
			_iState:=_iState+1;
			_ErrorState:=0;
			
		END_IF
	
	
	1:
		(*
		IF NOT _initError AND init  THEN
			InitDone:=TRUE; 
			 _iState:=_iState+1;
		END_IF
		*)	 
		IF init THEN 
			IF NOT _initError THEN
				InitDone:=TRUE;
				_iState:=_iState+1;	 
			ELSE
				Error:=TRUE;
				InitDone:=FALSE;
				_ErrorState:=_iState;
				nErrId_ADS:=_initADSErrorID;
				nFbErrorID:=_initFbErrorID;
				_initError:=FALSE;
				_iState:=0;		
			END_IF
		END_IF

	2:	
		 _iState:=_iState+1;
		
	3://Boxname
		GetBoxName();	
	
	4://Check the posibility of backup and restore 
				_EventTrigger(CLK:=TRUE);
		IF _EventTrigger.Q THEN 
			IF iAction=2 AND Servicetype=eSERVICE.Restore THEN 
				// File log restore action started
				_eventText:=CONCAT(CONCAT('Restore action of ',_sBoxName), ' is started');
				
			ELSIF iAction=0  THEN
				IF (Servicetype=eSERVICE.Backup OR Servicetype=eSERVICE.Backup_RevDocu) THEN  
					_eventText:=CONCAT(CONCAT('Backup action of ',_sBoxName), ' is started');
				ELSIF Servicetype=eSERVICE.Restore THEN 
					_eventText:=CONCAT(CONCAT('Restore action of ',_sBoxName), ' is started');
				END_IF	
			ELSE
				//error if action is restore action is shown and backup service is chosen by user and vice versa 
				_eventText:=CONCAT(_sBoxName, ' Read or write not possible, choose Service input according to iAction');
				 Error:=TRUE;
				 //Fehler code
				 nFbErrorID:=eFBERROR.WrongServiceTypeInput;
				 _ErrorState:=_iState;
			END_IF
			IF NOT Error THEN 
				_fbLogger.AddEvent(sEventText:=_eventText,EventType:='Info');
				_EventTrigger(CLK:=FALSE);	
				Error:=FALSE;
				_iState:=_iState+1;
			ELSE
				_fbLogger.AddEvent(sEventText:=_eventText,EventType:='Warning');
				_EventTrigger(CLK:=FALSE);	
				_iState:=0;
			END_IF
		END_IF	
	
	5://set call statement before activation of process 
		//TO-DO depending on the serviceType from user and iAction output set the commandline if there is a mismatch then log message 
		//Backup the project 
		IF Servicetype=eSERVICE.Backup THEN
			 _CommandLine:=GetCommandString();
			//Restore the project 
		ELSIF Servicetype=eSERVICE.Restore THEN 
			_CommandLine:=GetCommandString();
			//backup with reverse documentation 
		ELSIF Servicetype=eSERVICE.Backup_RevDocu THEN 
			_CommandLine:=GetCommandString();
		ELSE
			_CommandLine:='';	
		END_IF
		_iState:=_iState+1;
		
	6://Activate Process
		 ActivateProcess(); 
		
	
	7://Wait for Receiving flags or start monitoring timeout 
		_fbTimeOut.IN:=TRUE;
		IF NOT Done AND _fbTimeOut.Q THEN 
			Error:=TRUE;//Timeout
			_ErrorState:=_iState;
			 nFbErrorID:=eFBERROR.TimeoutExceed;
			_fbTimeOut.IN:=FALSE;
			//Event trigger 
			_ErrorMessage:=CONCAT4(STR1:=GetInstanceName(_spath),STR2:=' ',STR3:='Timeout ',STR4:='No Backup or restore posssible');
			_BackupRestoreTrig(CLK:=TRUE);
			IF _BackupRestoreTrig.Q THEN 
			_fbLogger.AddEvent(sEventText:=_ErrorMessage,EventType:='Error');
			_BackupRestoreTrig(CLK:=FALSE);				
			END_IF			
			_iState:=99;					
		ELSIF SynchronousFlagHandle(SynchronousValue:=TO_INT(_Synchronous_flag))=1 THEN 
				//Receive flag is high backup or restore is successful  
				_iState:=_iState+1;
		ELSIF SynchronousFlagHandle(SynchronousValue:=TO_INT(_Synchronous_flag))>1 THEN 
				Error:=TRUE;
				//error codes are handled in methods 
				_iState:=99;					
		END_IF	

	8:
		  IF Servicetype=eSERVICE.Restore THEN 
				_iState:=_iState+1;
		  ELSIF iAction=0 AND  (Servicetype=eSERVICE.Backup OR Servicetype=eSERVICE.Backup_RevDocu) THEN
				//log the file with backup successful
 				_eventText:=CONCAT(_sBoxName,' project backup successful');
				_BackupRestoreTrig(CLK:=TRUE);
				IF _BackupRestoreTrig.Q THEN 
					_fbLogger.AddEvent(sEventText:=_eventText,EventType:='Info');
					_BackupRestoreTrig(CLK:=FALSE);
				END_IF			
 				Done:=TRUE;
				_xFirstInvocation:=TRUE;
				Busy:=FALSE;
				_iState:=0;	
			END_IF
		
	9:(*when new slave address is added to the topology add entry in the Deviceinfo structure*)
		IF _newSlave_In_Topology  OR (_newFileCreated OR _nState_FileHandle=30)  THEN 
			(*Add new entry in the deviceinfo structure*)
			FOR i:=1 TO GVL_Constant.MAX_STOBER_SLAVES DO 
				IF GLOBAL_DeviceInfo.arr_DeviceInfodata[i].Slave_Address='' AND 
					GLOBAL_DeviceInfo.arr_DeviceInfodata[i].Production_Number='' THEN
					GLOBAL_DeviceInfo.arr_DeviceInfodata[i].Slave_Address:=TO_STRING(Slave_addr);
					GLOBAL_DeviceInfo.arr_DeviceInfodata[i].Production_Number:=_readDriveControllerProductionNr;
					_istate:=11;
					EXIT;
				END_IF	
			END_FOR
		ELSE
            _iState:=_istate+1;	
		END_IF
			
	10:(*Replace the production number in the deviceinfo structure array*)
		FOR _indexArray:=1 TO GVL_Constant.MAX_STOBER_SLAVES DO 
			IF GLOBAL_DeviceInfo.arr_DeviceInfodata[_indexArray].Slave_Address=TO_STRING(Slave_addr) THEN
				_oldProductionNr:=GLOBAL_DeviceInfo.arr_DeviceInfodata[_indexArray].Production_Number;
				GLOBAL_DeviceInfo.arr_DeviceInfodata[_indexArray].Production_Number:=_readDriveControllerProductionNr;
				_iState:=_iState+1;
				EXIT;
			END_IF
		END_FOR
		
	11:(*Prepare data*)	
		PrepareFileWriteData();
		
	12:(*Store the production number in the file*) 	
		(*open file in write mode and store the deviceinfo data structure array in file*) 
		_fbFileOpen(sNetId:='',sPathName:=_deviceDescPath ,nMode:=FOPEN_MODEWRITE OR FOPEN_MODETEXT ,ePath:=PATH_GENERIC ,bExecute:=TRUE , hFile=>_hFile );
			IF NOT _fbFileOpen.bBusy THEN 
				IF _fbFileOpen.bError THEN 
					_fbFileOpen(sNetId:='',bExecute:=FALSE);
					nErrId_ADS:=_fbFileOpen.nErrId;
					_ErrorMessage:=CONCAT4(STR1:=GetInstanceName(_spath),STR2:=' ',STR3:='ADS Error ',STR4:=TO_STRING(nErrId_ADS));
					Error:=TRUE;//Generate log 
					_ErrorState:=_iState;
					_fbFileOpen(sNetId:='',bExecute:=FALSE);
					_iState:=99;
				ELSE
					_fbFileOpen(sNetId:='',bExecute:=FALSE);
					_iState:=_iState+1;
				END_IF
			END_IF
	
	13:(*File write*)
		_fbFileWrite(sNetId:='',hFile:=_hFile,pWriteBuff:=ADR(_FileWriteByteArray),cbWriteLen:=GetSizeofFileWriteData(),bExecute:=TRUE,tTimeout:=T#5S );
		IF NOT _fbFileWrite.bBusy THEN 
				IF _fbFileWrite.bError THEN 
					_fbFileWrite(sNetId:='',bExecute:=FALSE);
					nErrId_ADS:=_fbFileWrite.nErrId;
					_ErrorMessage:=CONCAT4(STR1:=GetInstanceName(_spath),STR2:=' ',STR3:='ADS Error ',STR4:=TO_STRING(nErrId_ADS));
					Error:=TRUE;(*Generate log*) 
					_ErrorState:=_iState;
					_fbFileWrite(sNetId:='',bExecute:=FALSE);
					_iState:=99;
				ELSE
					_fbFileWrite(sNetId:='',bExecute:=FALSE);
					_iState:=_iState+1;
				END_IF
		END_IF
		
	14:(*close the file*)
			_fbFileClose(sNetId:='',hFile:=_hFile,bExecute:=TRUE);
			IF NOT _fbFileClose.bBusy THEN 
				IF _fbFileClose.bError THEN 
					nErrId_ADS:=_fbFileClose.nErrId;
					Error:=TRUE;
					_ErrorState:=_iState;
					_ErrorMessage:=CONCAT4(STR1:=GetInstanceName(_spath),STR2:=' ',STR3:='ADS Error ',STR4:=TO_STRING(nErrId_ADS));
					_fbFileClose(sNetId:='',bExecute:=FALSE);
					_iState:=99;
				ELSE
					_fbFileClose(sNetId:='',bExecute:=FALSE);	
					_iState:=_iState+1;
				END_IF
			END_IF
	 	
	15:(*new Production number is added*)
			_EventTrigger(CLK:=TRUE);
			IF iAction=2 THEN
				IF _oldProductionNr='' THEN 
					_eventText:=CONCAT8('New Slave ',TO_STRING(Slave_addr),' ', _sBoxName, ' with Prod.Nr. ', _readDriveControllerProductionNr ,' is added','');
				ELSE
					_eventText:=CONCAT8('Restore is successful ','Prod.Nr. ',_oldProductionNr,' is replaced with Prod.Nr. ',_readDriveControllerProductionNr, '','','');
				END_IF
				IF _EventTrigger.Q THEN 
					_fbLogger.AddEvent(sEventText:=_eventText,EventType:='Info');
					Done:=TRUE;
					_xFirstInvocation:=TRUE;
					Busy:=FALSE;	
					iAction:=0;	
					_iState:=0;		
				END_IF
			ELSIF iAction=0 THEN 
				Done:=TRUE;
				_xFirstInvocation:=TRUE;
				Busy:=FALSE;
				_iState:=0;	
			END_IF	
	
	99:(*Trigger event*) 	
		Error:=TRUE;
		_iState:=0;	
		
		
ELSE
		_iState:=0;
END_CASE
END_METHOD

METHOD PRIVATE CallInternalFbs : BOOL
VAR_INPUT
END_VAR
(*function block to check the file directory if exist*) 
	(*Project file path*) 
_fbFilepath_EnumFindFileEntry(sNetId:='' ,sPathName:=Filepath , eCmd:=E_EnumCmdType.eEnumCmd_First );
	(*DS6 process path*) 
_fbDS6ProcessPath_EnumFindFileEntry(sNetId:='' ,sPathName:=DS6_ProcessPath , eCmd:=E_EnumCmdType.eEnumCmd_First );

(*read boxname from the drive controller parameter A251*)
fbSdoReadBoxName(
				 sNetId:=AmsNetId_EtherCAT_Master , 
				 nSlaveAddr:=Slave_addr , 
				 nSubIndex:=16#0 , 
				 nIndex:=16#20FB , 
				 pDstBuf:=ADR(_sBoxName) , 
				 cbBufLen:=SIZEOF(_sBoxName)
				);

			

//Commandline later change with GetCommandString method 
(*_ActivateNTProcess(NETID:='' ,PATHSTR:='C:\Windows\py.exe' , 
            	   DIRNAME:='C:\Windows' , COMNDLINE:=Commandline);	*)			

//Activate the process				   
_ActivateNTProcess(NETID:='' ,PATHSTR:=CONCAT(DS6_ProcessPath,'\DS6A.exe') , 
            	   DIRNAME:=DS6_ProcessPath , COMNDLINE:=GetCommandString());
END_METHOD

METHOD PRIVATE GetADSPort : UINT
VAR_INPUT
END_VAR
GetADSPort:=TwinCAT_SystemInfoVarList._AppInfo.AdsPort;
END_METHOD

(*The method reads the Boxname of the Stober Slave device*)
METHOD PRIVATE GetBoxName : BOOL
//execute the function block fbSdoReadBoxName function block body is called in CallInternalFBs
fbSdoReadBoxName(bExecute:=TRUE);				
 			 
//TO-DO error check 
IF NOT fbSdoReadBoxName.bBusy THEN 
	
	IF fbSdoReadBoxName.bError THEN 
		Error:=TRUE;
		_ErrorState:=_iState;
		nErrId_ADS:=fbSdoReadBoxName.nErrId;
		fbSdoReadBoxName(bExecute:=FALSE);	
		_ErrorMessage:=Concat4(STR1:=GetInstanceName(_spath),STR2:=' ',STR3:='Boxname SDOread ADS Error ',STR4:=TO_STRING(nErrId_ADS));
		_BackupRestoreTrig(CLK:=TRUE);
		IF _BackupRestoreTrig.Q THEN 
			_fbLogger.AddEvent(sEventText:=_ErrorMessage,EventType:='Error');
			_BackupRestoreTrig(CLK:=FALSE);
		END_IF
		_iState:=99;	
		RETURN;
	END_IF
	//Check if BoxName is an empty string 
	IF _sBoxName='' THEN 
		Error:=TRUE;
		//Fehler code 107
		nFbErrorID:=eFBERROR.InvalidBoxname;
		_ErrorState:=_iState;
		_ErrorMessage:=Concat4(STR1:=GetInstanceName(_spath),STR2:=' ',STR3:='BoxName is empty ',STR4:='Boxname function block is not executed');
		fbSdoReadBoxName(bExecute:=FALSE);			
		_BackupRestoreTrig(CLK:=TRUE);
		IF _BackupRestoreTrig.Q THEN 
			_fbLogger.AddEvent(sEventText:=_ErrorMessage,EventType:='Error');
			_BackupRestoreTrig(CLK:=FALSE);
		END_IF
		_iState:=99;
	ELSE
		fbSdoReadBoxName(bExecute:=FALSE);	
		//STRING_TO_UTF8(pSrcSTRING:=ADR(_sBoxName),pDstUTF8:=ADR(_sBoxNameUTF_8),nDstSize:=SIZEOF(_sBoxNameUTF_8));
		_iState:=_iState+1;	
	END_IF
END_IF
END_METHOD

(*Method returns a commandline which is then used to send the DriveControlSuite application for the read or write of the project*)
METHOD PROTECTED GetCommandString : T_MaxString

VAR
	 {attribute 'TcEncoding':='UTF-8'}
	_CommandString:T_MaxString;
END_VAR
(*Start DS6 applicationfrom TwinCAT
Commandline=> DS6.exe -command <command> --boxname <Boxname> --productionnumber <number> --projectpath <path> --instancename <name>
*)
_projectPath:=Filepath;
IF Servicetype=eSERVICE.Backup THEN 
	_CommandString:=CONCAT4(STR1:=CONCAT4(STR1:=CONCAT8(
							STR1:='DS6A.exe ' , 
							STR2:='--command ' , 
							STR3:='backup ' , 
							STR4:='--boxname ' , 
							STR5:= concat('"', concat( _sBoxName,'"')) , 
							STR6:=' --productionnumber ' , 
							STR7:=_readDriveControllerProductionNr , 
							STR8:=' --projectpath ' ),
							STR2:=CONCAT('"',CONCAT(_projectPath,'"')),
							STR3:=' --instancename ',
							STR4:=SUPER^.GetInstanceName(_spath)	),
							STR2:='',STR3:='',STR4:='');
							
							
ELSIF Servicetype=eSERVICE.Backup_RevDocu THEN 
	_CommandString:=CONCAT4(STR1:=CONCAT4(STR1:=CONCAT8(
							STR1:='DS6A.exe ' , 
							STR2:='--command ' , 
							STR3:='backup_revdocu ' , 
							STR4:='--boxname ' , 
							STR5:= concat('"', concat( _sBoxName,'"')) , 
							STR6:=' --productionnumber ' , 
							STR7:=_readDriveControllerProductionNr , 
							STR8:=' --projectpath ' ),
							STR2:=CONCAT('"',CONCAT(_projectPath,'"')),
							STR3:=' --instancename ',
							STR4:=SUPER^.GetInstanceName(_spath)	),
							STR2:='',STR3:='',STR4:='');
							
							
ELSIF Servicetype=eSERVICE.Restore THEN 
	_CommandString:=CONCAT4(STR1:=CONCAT4(STR1:=CONCAT8(
							STR1:='DS6A.exe ' , 
							STR2:='--command ' , 
							STR3:='restore ' , 
							STR4:='--boxname ' , 
							STR5:= concat('"', concat(_sBoxName ,'"')) ,
							STR6:=' --productionnumber ' , 
							STR7:=_readDriveControllerProductionNr , 
							STR8:=' --projectpath ' ),
							STR2:=CONCAT('"',CONCAT(_projectPath,'"')),
							STR3:=' --instancename ',
							STR4:=SUPER^.GetInstanceName(_spath)),
							STR2:='',STR3:='',STR4:='');
END_IF	

//Return commandstring 
GetCommandString:=_CommandString;
END_METHOD

(*method to get the production number from the linetext of the Deviceinfo.txt file*)
METHOD PRIVATE GetProductionNumber : String
VAR_INPUT
	Str1	:STRING;
END_VAR
VAR
	ptByte		:POINTER TO BYTE;
	ptDestByte	:POINTER TO BYTE;
	ptrRtnByte	:POINTER TO BYTE;
	i			:INT;
	count		:INT;
	arrByte		:ARRAY [0..255] OF BYTE;
	j			:UINT;
END_VAR
//set the initial adress 
ptByte:=ADR(Str1);
ptDestByte:=ptByte;
//reset the Array of byte 
FOR j:=0 TO 255 DO 
	arrByte[j]:=0;
END_FOR
ptrRtnByte:=ADR(arrByte);//set initial adress 

count:=0;
FOR i:=0 TO LEN(Str1) DO 
	IF ptDestByte^<>0 THEN
		//save the string
		IF ptDestByte^=58 THEN  //check for ':' character 
			count:=count+1;
		END_IF 
		IF count>=2 THEN
			IF count=2 AND  ptDestByte^=58 THEN 
				ptDestByte:=ptDestByte+1;
			END_IF
			ptrRtnByte^:=ptDestByte^;//here start with ProdctionNr XXXXXX
			ptrRtnByte:=ptrRtnByte+1;
		END_IF
		ptDestByte:=ptDestByte+1;
	END_IF
END_FOR
//Replace $N with empty char in Bytearray
FOR j:=0 TO 255 DO 
	IF arrByte[j]=10 THEN //Ascii 10=$N(new line character 
		arrByte[j]:=0;
		exit;
	end_if
end_FOR


GetProductionNumber:=BYTEARR_TO_MAXSTRING(arrByte);
END_METHOD

METHOD PRIVATE GetSizeofFileWriteData : UDINT
VAR_INPUT
END_VAR

VAR
	i: INT;
	udi_countTotalByteArraySize:UDINT;
END_VAR
FOR i:=0 TO MAX_BYTEARRAY_SIZE DO 
	IF _FileWriteByteArray[i]<>0 THEN
		udi_countTotalByteArraySize:=udi_countTotalByteArraySize+1;
	END_IF
END_FOR

GetSizeofFileWriteData:=udi_countTotalByteArraySize;
END_METHOD

METHOD PRIVATE GetSlaveAddress : STRING
VAR_INPUT
	Str1:STRING;
END_VAR
VAR		
	ptByte		:POINTER TO BYTE;
	ptDestByte	:POINTER TO BYTE;
	ptrRtnByte	:POINTER TO BYTE;
	i			:INT;
	count		:INT;
	arrByte		:ARRAY [0..255] OF BYTE;
	j			:UINT;
	_SlaveAdrStart	:BOOL;
END_VAR
//set the initial adress 
ptByte:=ADR(Str1);
ptDestByte:=ptByte;
//reset the Array of byte 
FOR j:=0 TO 50 DO 
	arrByte[j]:=0;
END_FOR
ptrRtnByte:=ADR(arrByte);//set initial adress 

count:=0;
FOR i:=0 TO LEN(Str1) DO 
	IF ptDestByte^<>0 THEN
		//save the string
		IF ptDestByte^=58 THEN  //check for ':' character 
			_SlaveAdrStart:=TRUE;
			ptDestByte:=ptDestByte+1;
		END_IF
		IF _SlaveAdrStart THEN 
			IF ptDestByte^=59 THEN 
				EXIT;
			ELSE
				ptrRtnByte^:=ptDestByte^;
				ptrRtnByte:=ptrRtnByte+1;
			END_IF  
		END_IF
		ptDestByte:=ptDestByte+1;
	END_IF	
END_FOR

GetSlaveAddress:=BYTEARR_TO_MAXSTRING(arrByte);
END_METHOD

(*Method to handle function block output variable Done,Busy,Error*)
METHOD PRIVATE OutputHandle : BOOL
VAR_INPUT
	
END_VAR
VAR
	
END_VAR
(*At a time only one variale should be true after the rise trigger of execute*)
//if error is occured after execute
IF Error THEN 
	Busy:=FALSE;
END_IF
//reset error if no execute 
IF Error AND NOT Execute THEN 
	Error:=FALSE;
	nErrId_ADS:=0;
	nFbErrorID:=0;
END_IF
//Reset done if no execute
IF Done AND NOT Execute THEN
	Done:=FALSE; 
	_xFirstInvocation:=FALSE;
END_IF
END_METHOD

METHOD PRIVATE PrepareFileWriteData : BOOL
VAR_INPUT
END_VAR

VAR
	iByteArrayIndex				: INT;
	iStoberSlaveIndex			: INT;
	iFileLineIndex				: INT;
	DeviceInfoTextLineString	: STRING;
END_VAR
iByteArrayIndex:=0; 
FOR iStoberSlaveIndex:=1 TO GVL_Constant.MAX_STOBER_SLAVES DO
	
	IF GLOBAL_DeviceInfo.arr_DeviceInfodata[iStoberSlaveIndex].Slave_Address<>'' AND GLOBAL_DeviceInfo.arr_DeviceInfodata[iStoberSlaveIndex].Production_Number<>'' THEN 
	
		FOR iFileLineIndex:=0 TO LEN(SetFileLine(SlaveAddr:=GLOBAL_DeviceInfo.arr_DeviceInfodata[iStoberSlaveIndex].Slave_Address,ProdNr:=GLOBAL_DeviceInfo.arr_DeviceInfodata[iStoberSlaveIndex].Production_Number))-1 DO
			
			IF iByteArrayIndex<MAX_BYTEARRAY_SIZE THEN
				DeviceInfoTextLineString:=SetFileLine(SlaveAddr:=GLOBAL_DeviceInfo.arr_DeviceInfodata[iStoberSlaveIndex].Slave_Address,ProdNr:=GLOBAL_DeviceInfo.arr_DeviceInfodata[iStoberSlaveIndex].Production_Number);
				 _FileWriteByteArray[iByteArrayIndex]:=DeviceInfoTextLineString[iFileLineIndex];
				 IF iFileLineIndex<>LEN(SetFileLine(SlaveAddr:=GLOBAL_DeviceInfo.arr_DeviceInfodata[iStoberSlaveIndex].Slave_Address,ProdNr:=GLOBAL_DeviceInfo.arr_DeviceInfodata[iStoberSlaveIndex].Production_Number)) THEN 
				 	iByteArrayIndex:=iByteArrayIndex+1;
				 END_IF	
			END_IF
 		
		END_FOR
	ELSE
		_iState:=_iState+1;
		EXIT;	
	END_IF
	
END_FOR
END_METHOD

(*Method returns the linetext(slaveAdr:xxxx;ProdNr:xxxxxxx) which is stored in the Deviceinfo.txt file*)
METHOD PRIVATE SetFileLine : STRING
VAR_INPUT
	SlaveAddr	:STRING;
	ProdNr		:STRING;
END_VAR
VAR
	sFileLine	:STRING:='';
END_VAR
(*The slave address and production number that need to saved in the Deviceinfo.txt file
  e.g. SlaveAdr:1001;ProdNr:9001151 *)
sFileLine:=CONCAT(STR1:='SlaveAdr:',STR2:=TO_STRING(SlaveAddr));
sFileLine:=CONCAT(CONCAT(STR1:=sFileLine,STR2:=';'),STR2:='ProdNr:');
sFileLine:=Concat(STR1:=sFileLine,STR2:=ProdNr);
sFileLine:=CONCAT(STR1:=sFileLine,STR2:='$N');

//Return fileline 
SetFileLine:=sFileLine;
END_METHOD

METHOD PRIVATE SetTimeout : TIME
VAR_INPUT
END_VAR

VAR
	_Timeout: TIME;
END_VAR
IF Servicetype=eSERVICE.Backup OR Servicetype=eService.Backup_RevDocu THEN 
	_Timeout:=T#60S;
ELSIF Servicetype=eSERVICE.Restore THEN 
	_Timeout:=T#90S;	
ELSE
	_Timeout:=T#90S;	
END_IF

SetTimeout:=_Timeout;
END_METHOD

METHOD PRIVATE SynchronousFlagHandle : INT
VAR_INPUT
	SynchronousValue		:INT;
END_VAR


VAR
	ADS_ReturnValue:INT;
END_VAR
//TO-DO 
(*Method to handle Script mode return values*)
(*
	• Backup oder Restore ist erfolgreich------------------------------------------------------> 1
	• Drive controller project not found ------------------------------------------------------> 201
	• Drive controller project found several times in the project folder-----------------------> 203
	• Project open error ----------------------------------------------------------------------> 205	
	• Conncection to drive controller failed---------------------------------------------------> 207
	• Online connection failed ----------------------------------------------------------------> 209
*)	
ADS_ReturnValue:=SynchronousValue;

CASE ADS_ReturnValue OF 
	
	0:(*Default value do nothing*)
		SynchronousFlagHandle:=0;
		nFbErrorID:=eFBERROR.NoError;
		
	1:(*Backup or restore done*)
		SynchronousFlagHandle:=1;
		nFbErrorID:=eFBERROR.NoError;
		
	2:(*Drive controller project not found,Error code-201*)
		SynchronousFlagHandle:=2;
		nFbErrorID:=eFBERROR.ProjectNotFound;
															
	3:(*Drive Controller found several times in project,Error code-203*)
		SynchronousFlagHandle:=3;
		nFbErrorID:=eFBERROR.MoreThanOneProjectFound;
		
	4:(*Project open error, Error code-205*)
		SynchronousFlagHandle:=4;
		nFbErrorID:=eFBERROR.OpenProjectError;
		
	5:(*Connection to Drive controller failed,Error code-207*)
		SynchronousFlagHandle:=5;
		nFbErrorID:=eFBERROR.ConnectionError;
		
	6:(*Online connection failed ,Error code-209*)
		SynchronousFlagHandle:=6;
		nFbErrorID:=eFBERROR.OnlineError;
		
	7:
		SynchronousFlagHandle:=7;
		//nFbErrorID:=eERROR.DriveControllerConnnectionFailed;
		
	8:
		SynchronousFlagHandle:=8;
		//nFbErrorID:=eERROR.DriveControllerNotAccessible;
		
	9:
		SynchronousFlagHandle:=9;
		//nFbErrorID:=eERROR.ConfigurationReadFailed;
		
	10:
		SynchronousFlagHandle:=10;
		//nFbErrorID:=eERROR.ConfigurationWriteFailed;
		
	11:
		SynchronousFlagHandle:=11;
		//nFbErrorID:=eERROR.FailedToOpenProject;
		
	12:
		SynchronousFlagHandle:=12;
		//nFbErrorID:=eERROR.FailedToSaveProject;
ELSE
	SynchronousFlagHandle:=0;
END_CASE
END_METHOD

END_FUNCTION_BLOCK

// ---- POUs/STOBER_BoxName.TcPOU
{attribute 'hide_all_locals'}	
(*The function block write the STOBER Drive Device name from the EhterCAT IO Configuration 
 to the Drive parameter over EtherCAT SDO*)
FUNCTION_BLOCK STOBER_BoxName
VAR_INPUT
	AmsNetId_EtherCAT_Master:T_AmsNetID; (*AMS network identifier of the Ethercat master device*) 
	Execute:BOOL;		 (*Activates the block by a rising edge of this input *)
END_VAR
VAR_OUTPUT
	Error:BOOL;			(*Error is occured*)
	Busy:BOOL;			(*Function block is busy*)
	Done:BOOL;			(*Function block operation is successful*)
	ErrorID:UDINT;		(*Error ID*)
	FBErrorID:UDINT;	(*Function block ErrorID*)	
END_VAR
VAR

//Initialisation
	init:BOOL;
	Rtrig_Init:R_trig;
//Get Slave count method
	_Fb_GetSlaveCount:FB_EcGetSlaveCount;
	EC_MaxSlaves:UINT;
//Get the AMS network id method
	_sAmsNetID:T_AmsNetID;
//Get the ethercat master state method
	_FB_EcGetMasterState:FB_EcGetMasterState;
	_bSlaveConfigData: BOOL;
//Get slave config data 
	_FB_EcGetConfSlaves:FB_EcGetConfSlaves;
	_ArrEcConfSlaveInfo:ARRAY [0..GVL_Constant.MaxSlaves] OF ST_EcSlaveConfigData;
	_nStoeberSlaves:UINT;
//Get Slave devices 
	_arrStoeberDevices:ARRAY [0..GVL_Constant.MaxSlaves] OF StoeberSlavedesc;
	_StatechangeOld:ARRAY [0..GVL_Constant.MaxSlaves] OF INT;
//SDO write and slave state
	_FB_EcGetSlaveState:FB_EcGetSlaveState;
	_Fb_EtherCatWritePara: FB_EcCoESdoWrite;
	_bStatechanged:BOOL;
	iSlaveStateold:INT:=8;
	bAllSlaveInOpearation:BOOL;
	_Count: INT;
	_Ftrig:F_TRIG;
	SlavePreviousState:INT;
	iState:INT;
	_iIndex:UINT;
	_Windex:WORD;
	_iWrite:UINT;
//Act_SlaveStateChange
	i: INT;
	RS_State:RS;
	_R_Trig_SlaveStatus:R_Trig;
	_Execute_Trig	   :R_Trig;
	iLastErrorState:INT;
END_VAR

METH_StateMachine();
_Execute_Trig(CLK:=Execute);
METH_OutputHandle();

{attribute 'hide'}
METHOD METH_GetAMSID : BOOL
VAR_INPUT
END_VAR
//Falsche AMSnetID verknüft--Wrong AMSNetID connected
_sAmsNetID:=AmsNetId_EtherCAT_Master;
IF _sAmsNetID='' OR _sAmsNetID='0.0.0.0.0.0' THEN 
	Error:=TRUE;
	FBErrorID:=100; //'EtherCAT AMS ID is empty'
	//FBErrorID:=
	iLastErrorState:=iState;
	iState:=100;
ELSE	
	iState:=iState+1;
END_IF
END_METHOD

{attribute 'hide'}
METHOD METH_GetSlaveConfigData : BOOL
VAR_INPUT
END_VAR
VAR 
	fRtrig:R_Trig;
END_VAR
_FB_EcGetConfSlaves(
					sNetId:=_sAmsNetID , 
					pArrEcConfSlaveInfo:=ADR(_ArrEcConfSlaveInfo) , 
					cbBufLen:=SIZEOF(_ArrEcConfSlaveInfo) , 
					bExecute:=TRUE 
					);
					
IF NOT _FB_EcGetConfSlaves.bBusy THEN 
	_FB_EcGetConfSlaves.bExecute:=FALSE;
	IF _FB_EcGetConfSlaves.bError THEN 
		ErrorID:=_FB_EcGetConfSlaves.nErrorId;
		Error:=TRUE;
		Busy:=FALSE;
		iLastErrorState:=Istate;
		iState:=100;
	ELSE
		iState:=iState+1;	
	END_IF
END_IF
END_METHOD

{attribute 'hide'}
METHOD METH_GetSlaveCount : BOOL
VAR_INPUT
END_VAR
//Get all slave devices in configuration 
//Standard beckhoff function block to get the number of slaves in the device configuration
_Fb_GetSlaveCount(sNetId:=_sAmsNetID ,bExecute:= TRUE);
	
IF _Fb_GetSlaveCount.bExecute AND  NOT _Fb_GetSlaveCount.bBusy THEN 
	_Fb_GetSlaveCount(bExecute:=FALSE);
	IF 	_Fb_GetSlaveCount.bError THEN 
		EC_MaxSlaves:=0;
		Error:=TRUE;
		ErrorID:=_Fb_GetSlaveCount.nErrId;
		iLastErrorState:=iState;
		iState:=100;
	ELSE
		Error:=FALSE;
		EC_MaxSlaves:=_Fb_GetSlaveCount.nSlaves;
			IF  EC_MaxSlaves> GVL_Constant.MaxSlaves THEN 
				Error:=TRUE;
				FBErrorID:=200;
				Busy:=FALSE;
				iLastErrorState:=iState;
				iState:=100;
			ELSE
				iState:=iState+1;	
			END_IF
	END_IF
END_IF
//Number of actual slaves are more that defined constant
END_METHOD

{attribute 'hide'}
METHOD METH_GetSlaveDevices : BOOL
VAR_INPUT
END_VAR

VAR
	i:INT;
	j:INT;
	 //{attribute 'TcEncoding':='UTF-8'}
	destString:STRING(79);
END_VAR
VAR CONSTANT 
	_udiVendorID:UDINT:=185;
END_VAR
//Get Stoeber slave devices 
IF _bSlaveConfigData THEN
	j:=0;
	_nStoeberSlaves:=0;
	FOR i:=0 TO MIN(_FB_EcGetConfSlaves.nSlaves,GVL_Constant.MaxSlaves) DO 
		IF _ArrEcConfSlaveInfo[i].stSlaveIdentity.vendorId=_udiVendorID THEN 
		 _arrStoeberDevices[j].nAddr:=_ArrEcConfSlaveInfo[i].nAddr;
		 _arrStoeberDevices[j].nDevType:=_ArrEcConfSlaveInfo[i].nDevType;
		 //STRing_TO_UTF8(pSrcSTRING:=ADR(_ArrEcConfSlaveInfo[i].sName),pDstUTF8:=ADR(destString),nDstSize:=SIZEOF(destString));
		 _arrStoeberDevices[j].sName:=_ArrEcConfSlaveInfo[i].sName;
		  _arrStoeberDevices[j].sType:=_ArrEcConfSlaveInfo[i].sType;
		  j:=j+1;
		  _nStoeberSlaves:=_nStoeberSlaves+1;
		END_IF
	END_FOR
	iState:=iState+1;
END_IF
END_METHOD

{attribute 'hide'}
METHOD METH_GetSlaveState : BOOL
VAR_INPUT
END_VAR

VAR
	i: INT;
	j:INT;
END_VAR
//change of slave state when online 
j:=0;
SlavePreviousState:=_FB_EcGetSlaveState.state.deviceState;	
FOR i:=0 TO _nStoeberSlaves-1 DO 
	_StatechangeOld[i]:=_arrStoeberDevices[i].iState;
	_Label1:_FB_EcGetSlaveState(sNetId:=_sAmsNetID,
						nSlaveAddr:=_arrStoeberDevices[i].nAddr,
						bExecute:=TRUE);
//set error 					
	_arrStoeberDevices[i].iState:=_FB_EcGetSlaveState.state.deviceState	;	
	IF _FB_EcGetSlaveState.bBusy THEN
		JMP _Label1;
	ELSE	
		_FB_EcGetSlaveState(bExecute:=FALSE);			
	END_IF 		
	IF 	_StatechangeOld[i]<>_arrStoeberDevices[i].iState THEN 
		_bStatechanged:=TRUE;
	ELSE
		_bStatechanged:=FALSE;	
	END_IF 	
	IF _arrStoeberDevices[i].iState=8 THEN 
 		j:=j+1;
	END_IF
END_FOR

IF j=_nStoeberSlaves THEN 
	bAllSlaveInOpearation:=TRUE;
	iState:=iState+1;
ELSE
	bAllSlaveInOpearation:=FALSE;
	iLastErrorState:=iState;
	Error:=TRUE;
	FBErrorID:=300;
	iState:=100;
	Busy:=FALSE;
END_IF
//state change
END_METHOD

{attribute 'hide'}
METHOD METH_MasterState : BOOL
VAR_INPUT
END_VAR
_FB_EcGetMasterState(sNetId:=_sAmsNetID ,bExecute:=TRUE  );
	
IF NOT _FB_EcGetMasterState.bBusy THEN 
	_FB_EcGetMasterState(bExecute:=FALSE);
	IF _FB_EcGetMasterState.bError THEN 
		Error:=TRUE;
		ErrorID:=_FB_EcGetMasterState.nErrId;
		iLastErrorState:=iState;
		iState:=0;
	ELSE
		IF _FB_EcGetMasterState.state=INT_TO_WORD(Ethercat_State.PREOP)  OR 
			_FB_EcGetMasterState.state=INT_TO_WORD(Ethercat_State.OP) THEN 
			_bSlaveConfigData:=TRUE;
			iState:=iState+1;
		ELSE
			Error:=TRUE;
			FBErrorID:=400;
			_bSlaveConfigData:=FALSE;
			iState:=0;
		END_IF
	END_IF
END_IF
END_METHOD

METHOD PRIVATE METH_OutputHandle : BOOL
VAR_INPUT
END_VAR
(*At a time only one variale should be true after the rise trigger of execute*)
//if error is occured after execute
IF Error THEN 
	Busy:=FALSE;
END_IF
//reset error if no execute 
IF Error AND NOT Execute THEN 
	Error:=FALSE;
	ErrorID:=0;
	FBErrorID:=0;
END_IF
//Reset done if no execute
IF Done AND NOT Execute THEN 
	Done:=FALSE;
END_IF
END_METHOD

{attribute 'hide'}
METHOD METH_SlaveStateChange : BOOL
VAR_INPUT
END_VAR
IF FBErrorID=200 THEN 
	RETURN;
END_IF
//change of slave state when online 
SlavePreviousState:=_FB_EcGetSlaveState.state.deviceState;	
FOR i:=0 TO _nStoeberSlaves-1 DO 
	_StatechangeOld[i]:=_arrStoeberDevices[i].iState;
	_label1:_FB_EcGetSlaveState(sNetId:=_sAmsNetID,
						nSlaveAddr:=_arrStoeberDevices[i].nAddr,
						bExecute:=TRUE);
	//set error 					
_arrStoeberDevices[i].iState:=_FB_EcGetSlaveState.state.deviceState	;	
	IF 	_FB_EcGetSlaveState.bBusy THEN
		JMP _label1;	
	ELSE 
		_FB_EcGetSlaveState(bExecute:=FALSE);			
	END_IF 		
	IF 	_StatechangeOld[i]<>_arrStoeberDevices[i].iState  THEN 
		_bStatechanged:=TRUE;
	ELSE
		_bStatechanged:=FALSE;	
	END_IF
	//set when state is changed 
	RS_State(SET:=_bStatechanged);
END_FOR
// Trigger the Function block when slave state is changed
	_R_Trig_SlaveStatus(CLK:=RS_State.Q1);
	RS_State(RESET1:=_R_Trig_SlaveStatus.Q);
END_METHOD

METHOD PRIVATE METH_StateMachine : BOOL
VAR_INPUT
END_VAR
CASE iState OF 
//Check for the correct Ethercat AMS-NET ID 
	0:	
		_FB_EcGetConfSlaves(bExecute:=FALSE);
		_Fb_EtherCatWritePara(bExecute:=FALSE);
		IF _Execute_Trig.Q  THEN
			Error:=FALSE;
			Busy:=TRUE;
			Done:=FALSE;
			METH_GetAMSID();	
		END_IF
//Check the Ethercat master state 
	1:
		METH_MasterState();
//Get the slaves count in the topology 	
	2:
		METH_GetSlaveCount();
//Get the Ethercat slaves configuration data   	
	3:
		METH_GetSlaveConfigData();
//Filter out the stoeber Slaves data from the slave configuration data  		
	4:
		METH_GetSlaveDevices();
//Check the Ethercat slaves state connected in the hardware		
	5:
		METH_GetSlaveState();
//Write the Stoeber device name in the Drive Parameter A251	
	6:
		METH_WritePararmeter();	
//Error state 
	100://error state 
		//Execute:=FALSE;
		iState:=0;
END_CASE

//Action when the slave state is changed
END_METHOD

{attribute 'hide'}
METHOD METH_WritePararmeter : BOOL
VAR_INPUT
END_VAR
//Ethercat SDO Write  
//calculate the index of parameter A251 refer CiA402 manual (INDEX=(8192 +(GroupNO*512)+parameterNO))
//A251     _index:=8192+(0*512)+251;
_iIndex:=8192+(251);
_Windex:=UINT_TO_WORD(_iIndex);
_iWrite:=0;
_count:=0;

_Fb_EtherCatWritePara(	sNetId:=_sAmsNetID,nIndex:=_Windex ,nSubIndex:=0);
_FB_EcGetSlaveState(sNetId:=_sAmsNetID);						
FOR _iWrite:=0 TO (_nStoeberSlaves-1) DO 
		IF _arrStoeberDevices[_iwrite].iState=Ethercat_State.OP AND bAllSlaveInOpearation THEN 	
		_label1:	_Fb_EtherCatWritePara(nSlaveAddr:=_arrStoeberDevices[_iWrite].nAddr,
									pSrcBuf:=ADR(_arrStoeberDevices[_iWrite].sName),
									cbBufLen:=SIZEOF(_arrStoeberDevices[_iWrite].sName),
									bExecute:=TRUE);
			IF _Fb_EtherCatWritePara.bBusy THEN 
				JMP _label1;
			ELSIF _Fb_EtherCatWritePara.bError THEN 
				Error:=TRUE;
				ErrorID:=_Fb_EtherCatWritePara.nErrId;
				iState:=100;
				Busy:=FALSE;
			ELSE
				_Fb_EtherCatWritePara(bExecute:=FALSE);
				_FB_EcGetSlaveState(bExecute:=FALSE);
				_Count:=_Count+1;	
			END_IF
			
		END_IF 
END_FOR
	
IF _Count>=_nStoeberSlaves AND _iWrite>=_nStoeberSlaves THEN 
	Done:=TRUE;
	Busy:=FALSE;
	iState:=0;
ELSE
	iState:=0;
	Error:=TRUE;
END_IF
END_METHOD

END_FUNCTION_BLOCK

// ---- POUs/STOBER_MC_HOME.TcPOU
{attribute 'hide_all_locals'}
(*The function block executes the drive specific homing of the axis and saves the reference in the Drive contorller*)
FUNCTION_BLOCK STOBER_MC_HOME
VAR_INPUT
	Execute					:BOOL;				(*Start homing procedure with rising edge*)
	SetModeOfOperation		:SINT:=8;
END_VAR
VAR_OUTPUT
	Done					:BOOL;				(*Homing is done Successfully*)
	ModeOfOperation	AT %Q*	:SINT;				(*output of modes of operation to be linked to the drive PDO mapping*)
	Busy					:BOOL;				(*Homing procedure is active*)
	CommandAborted			:BOOL;				(*homing procedure was aborted*)
	Error					:BOOL;				(*Error is occured*)
	ErrorID					:UDINT;				(*Error ID*)
	FBErrorID				:eERROR;			(*Function block ErrorID*)
END_VAR
VAR
	_AxisStatus					:MC_ReadStatus;
	_stStatus					:ST_AxisStatus;
	_Drivedata					:MC_ReadDriveAddress;
	stdriveadress				:ST_DriveAddress;
	_PositionLagMonitor			:ADSWRITE;
	_ExecuteTrigger				:R_TRIG;
	istate						:INT;
	_LagMonitor					:UDINT;
	init						:BOOL;
	_writeNCIOOutput			:MC_WriteNcIoOutput;
	_WriteReferenceFlag			:ADSWRITE;
	_ReferenceFlag				:UDINT;
	_AdsSetPosition				:ADSWrite;
	_stSetPosition				:st_Set_Value;
	_HomeOffSet					:DINT;
	_fbHomeOffsetCOERead		:FB_CoERead;
	_IndexID_A569				:WORD;	
	_IndexID_A516				:WORD;
	_IndexID_A586				:WORD;
	_IndexID_A542				:WORD;
	_Active						:BOOL;
	_fbHomingMethodCOERead		:FB_CoERead;
	_HomingMethod				:DINT;
	_reloop						:BOOL;
	_statusloop					:BOOL;	
	_fbCOEStatusWord_Read		:FB_CoERead;
	_StatusWord					:DINT;
	_wStatusWord				:WORD;
	_fbCOE_ModeOfOpeationDisplay:FB_CoERead;
	_ModeOfOperationDisplay		:DINT;
END_VAR
VAR_IN_OUT
	Axis						:AXIS_REF;				(*reference to axis*)
END_VAR
VAR CONSTANT
	AXISA_A569_INDEX_ID			:WORD:=16#607C;
	AXISB_A569_INDEX_ID			:WORD:=16#687C;
	AXISA_A586_INDEX_ID			:WORD:=16#6098;
	AXISB_A586_INDEX_ID			:WORD:=16#6898;
	AXISA_A516_INDEX_ID			:WORD:=16#6041;
	AXISB_A516_INDEX_ID			:WORD:=16#6841;
	AXISA_A542_INDEX_ID			:WORD:=16#6061;
	AXISB_A542_INDEX_ID			:WORD:=16#6861;
	HOMING_MODE					:SINT:=6;
END_VAR

//Write mode of operation from user input on initialisation 
IF NOT init THEN 
	ModeOfOperation:=SetModeOfOperation;
	init:=TRUE;
END_IF
IF SetModeOfOperation<>8 AND SetModeOfOperation<>9 AND SetModeOfOperation<>10 AND Execute THEN 
	Error:=TRUE;
	FBErrorID:=eERROR.WRONG_MODE;
	RETURN;		
END_IF

M_InternFbCall();
M_StateMachine();
M_GetParameterIndex();
M_OutputHandle();
M_SetPosition();

//Write mode of operation from user input if homing run is not active
IF NOT _Active THEN 
	ModeOfOperation:=SetModeOfOperation;
END_IF

//Stop the homing run if axis error comes 
IF (_AxisStatus.Error OR _AxisStatus.ErrorStop) AND _Active THEN 
	iState:=0;
	ModeOfOperation:=SetModeOfOperation;
	Error:=TRUE;
	Busy:=FALSE;
	Done:=FALSE;
	_Active:=FALSE;
END_IF

METHOD PRIVATE M_GetParameterIndex : BOOL
VAR_INPUT
END_VAR
IF stdriveadress.Channel=0 THEN 
	_IndexID_A569:=AXISA_A569_INDEX_ID;//index id for parameter A569 Axis A
	_IndexID_A586:=AXISA_A586_INDEX_ID;//index id for parameter A586 Axis A
	_IndexID_A516:=AXISA_A516_INDEX_ID;//index id for parameter A541 Axis A
	_IndexID_A542:=AXISA_A542_INDEX_ID;//index id for parameter A542 Axis A
ELSIF stdriveadress.Channel=1 THEN 
 	_IndexID_A569:=AXISB_A569_INDEX_ID;//index id for parameter A569 Axis B
	_IndexID_A586:=AXISB_A586_INDEX_ID;//Index id for parameter A586 Axis B
	_IndexID_A516:=AXISB_A516_INDEX_ID;//Index id for parameter A541 Axis B
	_IndexID_A542:=AXISB_A542_INDEX_ID;//index id for parameter A542 Axis B
END_IF
END_METHOD

METHOD PRIVATE M_InternFbCall : BOOL
VAR_INPUT
END_VAR
{warning disable C0371}	
//Read axis status 
M_ReadStatus();
//Refer to twincat NC-ADS manual index group and index offset used below in the function blocks input 
//Get Drive NC-ADS access data 
_Drivedata(	Execute:=Execute,Axis:=Axis,DriveAddress=>stdriveadress );

//Rise trigger execute trigger for function block execution 	
_ExecuteTrigger(CLK:=Execute);
	
//Enable/Disable position lag monitoring 
_PositionLagMonitor(NETID:= ,Port:=501,IDXGRP:=16#6000+stdriveadress.NcAxisId,
				IDXOFFS:=16#10,LEN:=SIZEOF(_LagMonitor),SRCADDR:=ADR(_LagMonitor),TMOUT:=T#0.1S );
				
//Overwrite NC process image--> NC control word Ctrl1			
_writeNCIOOutput(Axis:=Axis ,Device:=E_NcIoDevice.NcIoDeviceDrive , 
	NcIoOutput:=E_NcIoOutput.NcIoOutputnCtrl1,BitSelectMask:=16#10 );			

//Set reset reference flag
_WriteReferenceFlag(NETID:='',PORT:=501,IDXGRP:=16#4200+stdriveadress.NcAxisId,
					IDXOFFS:=16#1B,LEN:=SIZEOF(_ReferenceFlag),SRCADDR:=ADR(_ReferenceFlag));	

//Set target postion 
_AdsSetPosition(NETID:='',PORT:=501,IDXGRP:=16#4100+stdriveadress.NcAxisId,
				IDXOFFS:=16#60,LEN:=SIZEOF(_stSetPosition),SRCADDR:=ADR(_stSetPosition));	
				
//Read homing methods
_fbHomingMethodCOERead(	NetId:='' ,Index:=_IndexID_A586,SubIndex:=0,pDstBuf:=ADR(_HomingMethod), 
						BufLen:=SIZEOF(_HomingMethod),Axis:= Axis);	
								
//Read status word A516
_fbCOEStatusWord_Read(NetId:='',Index:=_IndexID_A516,SubIndex:=16#0,Axis:=Axis,pDstBuf:=ADR(_StatusWord),
					 BufLen:=SIZEOF(_StatusWord));
											
//Read homing offset 
_fbHomeOffsetCOERead(NetId:= ,Index:=_IndexID_A569 ,SubIndex:=0 ,pDstBuf:= ADR(_HomeOffSet),
					 BufLen:=SIZEOF(_HomeOffSet) ,Axis:= Axis);		

//Read mode of operation display 
_fbCOE_ModeOfOpeationDisplay(NetId:='',Index:=_IndexID_A542,SubIndex:=0,pDstBuf:=ADR(_ModeOfOperationDisplay),
							 BufLen:=SIZEOF(_ModeOfOperationDisplay),Axis:=Axis);
END_METHOD

METHOD PRIVATE M_OutputHandle : BOOL
VAR_INPUT
END_VAR
//Reset Error when no Execute 
IF Error AND NOT Execute THEN 
	Error:=FALSE;
	ErrorId:=0;
	FBErrorID:=eERROR.NO_ERROR;
END_IF
//Reset Done if no execute 
IF Done AND NOT Execute THEN 
	Done:=FALSE;
END_IF
//Reset Commandaborted if no execute 
IF CommandAborted AND NOT Execute THEN 
	CommandAborted:=FALSE;
END_IF
END_METHOD

METHOD PRIVATE M_ReadStatus : BOOL
VAR_INPUT
END_VAR
{warning disable C0371}	
_AxisStatus(Axis:=Axis,Enable:=TRUE,Status=>_stStatus);
//check for motion command lock when homing is runnig and MC_Stop is executed then homing run is aborted
IF _stStatus.MotionCommandsLocked AND Busy THEN 
	CommandAborted:=TRUE;
	Busy:=FALSE;
	ModeOfOperation:=SetModeOfOperation;
	iState:=0;
END_IF

//Read the staus word A516 cyclic
IF busy AND iState>30 THEN 
	REPEAT 
		_statusloop:=FALSE;
		_fbCOEStatusWord_Read(Execute:=TRUE,Axis:=Axis);
		IF NOT _fbCOEStatusWord_Read.Busy THEN 
			_fbCOEStatusWord_Read(Execute:=FALSE,Axis:=Axis);
		END_IF
		IF  _fbCOEStatusWord_Read.Error THEN 
			_fbCOEStatusWord_Read(Execute:=FALSE,Axis:=Axis);
			Error:=TRUE;
			ErrorID:=_fbCOEStatusWord_Read.AdsErrId;
			iState:=900;
			EXIT;
		END_IF		
		
	UNTIL NOT _statusloop
	END_REPEAT
ELSE 
	_fbCOEStatusWord_Read(Execute:=FALSE,Axis:=Axis);	
END_IF

//abort command if axis enable is withdrawn during homing run 
_wStatusWord:=DINT_TO_WORD(_StatusWord);
IF Busy AND _wStatusWord.1=FALSE AND iState>50 THEN 
	CommandAborted:=TRUE;
	Busy:=FALSE;
	ModeOfOperation:=SetModeOfOperation;
	iState:=0;
END_IF
END_METHOD

METHOD PRIVATE M_SetPosition : BOOL
VAR_INPUT
END_VAR

VAR
	
END_VAR
{warning disable C0371}	
//Write target position during homing mode 
IF Busy AND iState>50 THEN 
	REPEAT 
		_reloop:=FALSE;
		_stSetPosition.SetPosition:=Axis.NcToPlc.ActPos;
		
		_AdsSetPosition(WRITE:=TRUE);
		IF NOT _AdsSetPosition.busy THEN 
			_AdsSetPosition(WRITE:=FALSE);
		END_IF
		IF _AdsSetPosition.ERR THEN 
			Error:=TRUE;
			ErrorID:=_AdsSetPosition.ERRID;
			iState:=900;
			EXIT;
		END_IF
	UNTIL NOT _reloop
	END_REPEAT	
END_IF
END_METHOD

METHOD PRIVATE M_StateMachine : BOOL
VAR_INPUT
END_VAR
{warning disable C0371}	
CASE istate OF 
	0://Reset all outputs 
		_Drivedata(Axis:=Axis,Execute:=FALSE);
		IF _ExecuteTrigger.Q THEN 
			IF _AxisStatus.Standstill THEN 
				_writeNCIOOutput.Execute:=FALSE;
				_AdsSetPosition(WRITE:=FALSE);
				_PositionLagMonitor(WRITE:=FALSE);
				_WriteReferenceFlag(WRITE:=FALSE);
				_fbHomingMethodCOERead(Axis:=Axis,Execute:=FALSE);
				_fbHomeOffsetCOERead(Execute:=FALSE ,Axis:= Axis);
				_WriteReferenceFlag(WRITE:=FALSE);	
				_fbCOEStatusWord_Read(Axis:=Axis,Execute:=FALSE);		
				Busy:=TRUE;
				_Active:=TRUE;
				Done:=FALSE;
				Error:=FALSE;
				ErrorID:=0;
				FBErrorID:=(eERROR.NO_ERROR);
				CommandAborted:=FALSE;
				iState:=iState+5;	
			ELSE
				Error:=TRUE;
				FBErrorID:=(eERROR.AXIS_NOT_ENABLED);
				istate:=900;	
			END_IF
		END_IF
	5://reset NC reference FLAG 
		_ReferenceFlag:=0;
		_WriteReferenceFlag(WRITE:=TRUE);
		IF NOT _WriteReferenceFlag.BUSY THEN 
			_WriteReferenceFlag(WRITE:=FALSE);
			iState:=iState+5;
		ELSIF _WriteReferenceFlag.ERR THEN
			Error:=TRUE;
			ErrorID:=_WriteReferenceFlag.ERRID;
			iState:=900;	
		END_IF
	
	10://Get the drive NC-ADS data 
		_Drivedata.Execute:=TRUE;
		IF NOT _Drivedata.Busy AND _Drivedata.Done THEN
			iState:=iState+10;
		END_IF 	
		IF _Drivedata.Error THEN 
			Error:=TRUE;
			iState:=900;
		END_IF
		
	20://Disable Position lag monitoring
		_LagMonitor:=0;
		_PositionLagMonitor(WRITE:=TRUE);
		IF NOT 	_PositionLagMonitor.BUSY THEN
			_PositionLagMonitor(WRITE:=FALSE);
			iState:=iState+10;
		ELSIF 	_PositionLagMonitor.ERR THEN 
			Error:=TRUE;
			ErrorID:=_PositionLagMonitor.ERRID;
			iState:=900;
		END_IF
		
	30: //set Mode of operation to homing mode 
			ModeOfOperation:=HOMING_MODE;	
			istate:=istate+10;
		
	40://confirm mode of operation 	
		_fbCOE_ModeOfOpeationDisplay(Execute:=TRUE,Axis:=Axis);
		IF NOT _fbCOE_ModeOfOpeationDisplay.Busy THEN 
			_fbCOE_ModeOfOpeationDisplay(Execute:=FALSE,Axis:=Axis);
			IF _ModeOfOperationDisplay<>HOMING_MODE THEN 
				Error:=TRUE;
				FBErrorID:=eERROR.NO_DEVICE_LINK;
				iState:=900;
			ELSE
				iState:=iState+10;	
			END_IF
		ELSIF 	_fbCOE_ModeOfOpeationDisplay.Error THEN 
			Error:=TRUE;
			ErrorID:=_fbCOE_ModeOfOpeationDisplay.AdsErrId;
			_fbCOE_ModeOfOpeationDisplay(Execute:=FALSE,Axis:=Axis);
			iState:=900;
		END_IF
		
			
	50://Read Homing offset 
		_fbHomeOffsetCOERead(Axis:=Axis,Execute:=TRUE);
		IF NOT _fbHomeOffsetCOERead.Busy THEN 
			_fbHomeOffsetCOERead(Execute:=FALSE ,Axis:= Axis);
			istate:=istate+10;
		ELSIF _fbHomeOffsetCOERead.Error THEN 
			Error:=TRUE;
			ErrorID:=_fbHomeOffsetCOERead.AdsErrId;
			iState:=900;
		END_IF
		
	60://Read homing method 
		_fbHomingMethodCOERead(Axis:=Axis,Execute:=TRUE);			
		IF NOT _fbHomingMethodCOERead.Busy THEN 
			_fbHomingMethodCOERead(Axis:=Axis,Execute:=FALSE);
			IF (_HomingMethod=0) THEN 
				Error:=TRUE;
				FBErrorID:=(eERROR.HOMING_METHOD_INACTIVE);
				iState:=900;
			ELSE	
				iState:=iState+10;	
			END_IF
		ELSIF 	_fbHomingMethodCOERead.Error THEN
			Error:=TRUE;
			ErrorID:=_fbHomingMethodCOERead.AdsErrId;
			iState:=900;
		END_IF
	70://Reset bit 4 of NC control word and start homing
		_writeNCIOOutput.BitValues:=0;
		_writeNCIOOutput.Execute:=TRUE;
		IF _writeNCIOOutput.Done THEN
				istate:=istate+10;
				_writeNCIOOutput.Execute:=FALSE;
		END_IF		
			
	80://wait till homing is done 	or wait till bit 10 of status word is true 	
		 IF _wStatusWord.10 = TRUE AND _wStatusWord.12 THEN 
			 ModeOfOperation:=8;
			 iState:=iState+10;
		 END_IF
		
	90://Set NC reference FLAG
		 _ReferenceFlag:=1;
		_WriteReferenceFlag(WRITE:=TRUE);
		IF NOT _WriteReferenceFlag.BUSY THEN 
			_WriteReferenceFlag(WRITE:=FALSE);
			iState:=iState+10;
		ELSIF _WriteReferenceFlag.ERR THEN
			Error:=TRUE;
			ErrorID:=_WriteReferenceFlag.ERRID;
			iState:=900;	
		END_IF
	100://Enable position monitoring 
		_LagMonitor:=1;
		_PositionLagMonitor(WRITE:=TRUE);
		IF NOT 	_PositionLagMonitor.BUSY THEN
			_PositionLagMonitor(WRITE:=FALSE);
			iState:=iState+10;
		ELSIF 	_PositionLagMonitor.ERR THEN 
			Error:=TRUE;
			ErrorID:=_PositionLagMonitor.ERRID;
		END_IF	
	
	110://set mode of operation back to setoperationmode 
		ModeOfOperation:=SetModeOfOperation;
		_writeNCIOOutput.BitValues:=0;
		_writeNCIOOutput.Execute:=TRUE;
		IF _writeNCIOOutput.Done THEN 
				_writeNCIOOutput.Execute:=FALSE;
				Done:=TRUE;
				Busy:=FALSE;
				_Active:=FALSE;
				iState:=0;
		END_IF
	
	900://Error state
		istate:=0;
		ModeOfOperation:=SetModeOfOperation;
		Busy:=FALSE;
		_Active:=FALSE;
END_CASE
END_METHOD

END_FUNCTION_BLOCK

// ---- Project Information/F_GetCompany.TcPOU
// This function has been automatically generated from the project information.
{attribute 'signature_flag' := '1073741824'}
{attribute 'TcGenerated'}
{attribute 'no-analysis'}
FUNCTION F_GetCompany : WSTRING
VAR_INPUT
	
END_VAR

F_GetCompany := "STÖBER Antriebstechnik GmbH + Co. KG";

END_FUNCTION

// ---- Project Information/F_GetTitle.TcPOU
// This function has been automatically generated from the project information.
{attribute 'signature_flag' := '1073741824'}
{attribute 'TcGenerated'}
{attribute 'no-analysis'}
FUNCTION F_GetTitle : WSTRING
VAR_INPUT
	
END_VAR

F_GetTitle := "STOBER_G6_Util";

END_FUNCTION

// ---- Project Information/F_GetVersion.TcPOU
// This function has been automatically generated from the project information.
{attribute 'signature_flag' := '1073741824'}
{attribute 'TcGenerated'}
{attribute 'no-analysis'}
FUNCTION F_GetVersion : ST_LibVersion
VAR_INPUT
	
END_VAR

F_GetVersion.iMajor := 3;
F_GetVersion.iMinor := 1;
F_GetVersion.iBuild := 1;
F_GetVersion.iRevision := 0;

END_FUNCTION
